FUNCTION RFID_Get_Bool : Buffer_Error
VAR_INPUT
	Data : REFERENCE TO RFID_Tag_Data;
	Num : USINT; 
END_VAR
VAR_IN_OUT
	Out : BOOL;
END_VAR

RFID_Get_Bool := Get_Bool_From_Buffer(Num:= Num, 
									Layout:= Data.Layout, 
									Buffer:= Data.Data, 
									Out:= Out);

END_FUNCTION

(* stored: Version 1.1.0.1, ProductVersion 3.1.4024.10
   POU RFID_Get_Bool: Id {dfceaa5d-6077-4deb-b6f7-508e955400ff}, SpecialFunc None *)
